FUNCTION_BLOCK PUBLIC FB_VISU_GATE_LOCK
VAR_INPUT
END_VAR
VAR_OUTPUT
END_VAR
VAR
	itfOpMode:												I_OP_MODE;
	itfUser:												I_USER_MANAGER;
	bClickGateLock:											BOOL;
	itfGateLock:											I_GATE_LOCK;	
	
	bEnable:												BOOL;
	bAdmin:													BOOL;
	sObjName:												STRING;
END_VAR

//Tastensperre bei Auto oder Keiner Betriebsartenauswahl
IF THIS^.itfOpMode.P_OP_MODE_STATE=OP_MODE.MANUAL THEN
	bEnable:=TRUE;
ELSE
	bEnable:=FALSE;
END_IF

bAdmin:=FALSE;
IF itfUser.P_UserGroupID=USER.Admin THEN
	bAdmin:=TRUE;
END_IF

METHOD FB_init : BOOL
VAR_INPUT
	bInitRetains : BOOL; // if TRUE, the retain variables are initialized (warm start / cold start)
	bInCopyCode : BOOL;  // if TRUE, the instance afterwards gets moved into the copy code (online change)
	itfOpMode:												I_OP_MODE;
	itfUser:												I_USER_MANAGER;
	itfDoorLock:											I_GATE_LOCK;
END_VAR
END_METHOD

END_FUNCTION_BLOCK

(* stored: Version 1.1.0.1, ProductVersion 3.1.4024.12
   POU FB_VISU_GATE_LOCK: Id {ddb62b23-3d27-4aa9-aeb0-22738384995a}, SpecialFunc None
   Method FB_init: Id {908cf542-b53e-4adb-a635-b1e6022ff4f9} *)
